TYPE unMyUINT :
UNION
	nUINT	: UINT;
	nUSINT	: ARRAY[1..2] OF USINT;
END_UNION
END_TYPE

(* stored: Version 1.1.0.1, ProductVersion 3.1.4024.12
   DUT unMyUINT: Id {5a80992d-e0e2-4bd8-a183-45c910ee8ea6} *)
